(* PLC project steel-plant, Generated TextualNotationConverter 1.0 *)
(* stored: creationDateTime 2025-07-30T12:00:00, modificationDateTime 2025-01-30T12:00:00 *)

FUNCTION_BLOCK ANALOG_IN
  VAR_INPUT
    Name : STRING;
    Description : STRING;
    Raw_Signal : REAL;
    PV_High : REAL;
    PV_Low : REAL;
    Scaling_Slope : REAL;
    Scaling_Offset : REAL;
    Alarm_Enable : BOOL;
  END_VAR
  VAR_OUTPUT
    PV : REAL;
    High_Alarm : BOOL;
    Low_Alarm : BOOL;
    General_Fault : BOOL;
  END_VAR

            
          
END_FUNCTION_BLOCK

FUNCTION_BLOCK PID_BASIC
  VAR_INPUT
    Name : STRING;
    Description : STRING;
    AUTO : BOOL;
    PV : REAL;
    SP : REAL;
    MV_MIN : REAL;
    MV_MAX : REAL;
    X0 : REAL;
    KP : REAL;
    TR : REAL;
    TD : REAL;
    PV_High : REAL;
    PV_Low : REAL;
    Deviation_Limit : REAL;
    Inhibit : BOOL;
  END_VAR
  VAR_OUTPUT
    PV_High_Alarm : BOOL;
    PV_Low_Alarm : BOOL;
    Deviation_Alarm : BOOL;
    XOUT : REAL;
  END_VAR

            
          
END_FUNCTION_BLOCK

FUNCTION_BLOCK RATIO_CONTROL
  VAR_INPUT
    Name : STRING;
    Description : STRING;
    Auto : BOOL;
    PrimaryPV : REAL;
    SecondaryPV : REAL;
    RatioSP : REAL;
    Bias : REAL;
    TrimKp : REAL;
    TrimTi : STRING;
    MV_MIN : REAL;
    MV_MAX : REAL;
    ManOut : REAL;
    Inhibit : BOOL;
  END_VAR
  VAR_OUTPUT
    SlaveSP : REAL;
    ActiveRatio : REAL;
    RatioErr : REAL;
  END_VAR

            
          
END_FUNCTION_BLOCK

FUNCTION_BLOCK VALVE_ELECTRIC
  VAR_INPUT
    Name : STRING;
    Description : STRING;
    Control_Signal : REAL;
    Manual_Mode : BOOL;
    Manual_Position : REAL;
    Open_Limit : REAL;
    Close_Limit : REAL;
    Timeout : STRING;
    Inhibit : BOOL;
  END_VAR
  VAR_OUTPUT
    Valve_Position : REAL;
    Feedback_Pos : REAL;
    Valve_Moving : BOOL;
    Position_Error : BOOL;
    Alarm : BOOL;
  END_VAR

            
          
END_FUNCTION_BLOCK

PROGRAM Section2
  VAR
    FT101_WildFlow_PV : REAL;
    FT102_FluxFlow_PV : REAL;
    TIT101_Temperature_PV : REAL;
    FFIC103_FluxFlowSP : REAL;
    FIC102_ValveCommand : REAL;
  END_VAR
  VAR
    FT-101 : ANALOG_IN;
    FT-102 : ANALOG_IN;
    TIT-101 : ANALOG_IN;
    FV-102 : VALVE_ELECTRIC;
    FIC-102 : PID_BASIC;
    FFIC-103 : RATIO_CONTROL;
  END_VAR
  VAR  (* added by the conversion: wires and edge detectors of the diagram *)
    _OR1_OUT : BOOL;
    _NOT2_OUT : BOOL;
  END_VAR

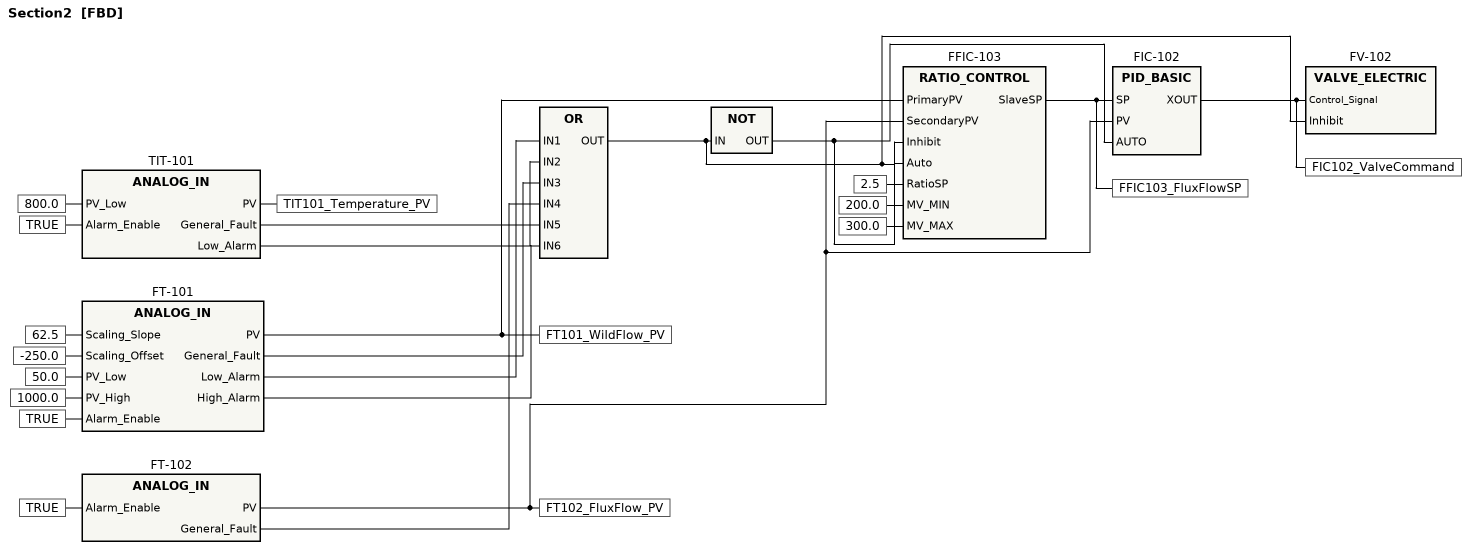
(* FBD diagram, written out as Structured Text *)
FT-101(Scaling_Slope := 62.5, Scaling_Offset := -250.0, PV_Low := 50.0, PV_High := 1000.0, Alarm_Enable := TRUE);
FT-102(Alarm_Enable := TRUE);
TIT-101(PV_Low := 800.0, Alarm_Enable := TRUE);
_OR1_OUT := FT-101.Low_Alarm OR TIT-101.Low_Alarm OR FT-101.General_Fault OR FT-102.General_Fault OR TIT-101.General_Fault OR FT-101.High_Alarm;
_NOT2_OUT := NOT _OR1_OUT;
FFIC-103(PrimaryPV := FT-101.PV, SecondaryPV := FT-102.PV, Inhibit := _OR1_OUT, Auto := _NOT2_OUT, RatioSP := 2.5, MV_MIN := 200.0, MV_MAX := 300.0);
FFIC103_FluxFlowSP := FFIC-103.SlaveSP;
FIC-102(SP := FFIC-103.SlaveSP, PV := FT-102.PV, AUTO := _NOT2_OUT);
FIC102_ValveCommand := FIC-102.XOUT;
FT101_WildFlow_PV := FT-101.PV;
FT102_FluxFlow_PV := FT-102.PV;
TIT101_Temperature_PV := TIT-101.PV;
FV-102(Control_Signal := FIC-102.XOUT, Inhibit := _OR1_OUT);
END_PROGRAM

FUNCTION_BLOCK BOOL_IN
  VAR_INPUT
    Name : STRING;
    Description : STRING;
    Bool_In : BOOL;
    Alarm_OnTrue : BOOL;
    Alarm_OnFalse : BOOL;
    Latch_Enable : BOOL;
    Reset_Latch : BOOL;
  END_VAR
  VAR_OUTPUT
    Bool_Out : BOOL;
    Alarm_Active : BOOL;
    Latched_Status : BOOL;
  END_VAR

            
          
END_FUNCTION_BLOCK

FUNCTION_BLOCK DIGITAL_IN
  VAR_INPUT
    Name : STRING;
    Description : STRING;
    DI_Raw : BOOL;
    DebounceTime : STRING;
    EnableAlarm : BOOL;
  END_VAR
  VAR_OUTPUT
    DI_Out : BOOL;
    Fault_State : BOOL;
  END_VAR

            
          
END_FUNCTION_BLOCK

FUNCTION_BLOCK DUTY_STANDBY
  VAR_INPUT
    Name : STRING;
    Description : STRING;
    Enable : BOOL;
    StartRequest : BOOL;
    AlternateEnable : BOOL;
    ForcePumpA : BOOL;
    ForcePumpB : BOOL;
    DutyElapsed : BOOL;
    MinRunElapsed : BOOL;
    SwitchoverDelayElapsed : BOOL;
    StartTimeoutElapsed : BOOL;
    PumpA_RunFB : BOOL;
    PumpB_RunFB : BOOL;
    PumpA_Fault : BOOL;
    PumpB_Fault : BOOL;
    Reset : BOOL;
    Inhibit : BOOL;
  END_VAR
  VAR_OUTPUT
    CmdPumpA : BOOL;
    CmdPumpB : BOOL;
    ActiveIsA : BOOL;
    SwitchedDueToDuty : BOOL;
    SwitchedDueToFailure : BOOL;
    Alarm_FailedStart_A : BOOL;
    Alarm_FailedStart_B : BOOL;
    Alarm_NoAvailablePump : BOOL;
  END_VAR

            
          
END_FUNCTION_BLOCK

FUNCTION_BLOCK MOTOR_2SPD
  VAR_INPUT
    Name : STRING;
    Description : STRING;
    Start_Cmd : BOOL;
    Stop_Cmd : BOOL;
    Speed_High_Cmd : BOOL;
    Speed_Low_Cmd : BOOL;
    Inhibit : BOOL;
  END_VAR
  VAR_OUTPUT
    Motor_Start_Out : BOOL;
    FB_Running : BOOL;
    FB_Trip : BOOL;
    FB_HighSpeed : BOOL;
    FB_LowSpeed : BOOL;
    Alarm_Speed_Error : BOOL;
  END_VAR

            
          
END_FUNCTION_BLOCK

FUNCTION_BLOCK MOTOR_ON_OFF
  VAR_INPUT
    Name : STRING;
    Description : STRING;
    Start_Cmd : BOOL;
    Stop_Cmd : BOOL;
    Start_Delay : STRING;
    MinRunTime : STRING;
    Inhibit : BOOL;
  END_VAR
  VAR_OUTPUT
    Motor_Start_Out : BOOL;
    FB_Running : BOOL;
    FB_Trip : BOOL;
    Alarm_Start_Fail : BOOL;
    Alarm_Stop_Fail : BOOL;
  END_VAR

            
          
END_FUNCTION_BLOCK

FUNCTION_BLOCK MOTOR_VSD
  VAR_INPUT
    Name : STRING;
    Description : STRING;
    Start_Cmd : BOOL;
    Stop_Cmd : BOOL;
    Speed_SP : REAL;
    Accel_Ramp : STRING;
    Decel_Ramp : STRING;
    Inhibit : BOOL;
  END_VAR
  VAR_OUTPUT
    Speed_Out : REAL;
    FB_Running : BOOL;
    FB_Fault : BOOL;
    FB_Ready : BOOL;
    FB_ActualSpeed : REAL;
    Alarm_Speed_Deviation : BOOL;
    Alarm_Comm_Fail : BOOL;
  END_VAR

            
          
END_FUNCTION_BLOCK

FUNCTION_BLOCK SPLIT_RANGE
  VAR_INPUT
    Name : STRING;
    Description : STRING;
    IN : REAL;
    Split_Point : REAL;
    Output1_Start : REAL;
    Output1_End : REAL;
    Output2_Start : REAL;
    Output2_End : REAL;
  END_VAR
  VAR_OUTPUT
    OUT1 : REAL;
    OUT2 : REAL;
  END_VAR

            
          
END_FUNCTION_BLOCK

FUNCTION_BLOCK VALVE_ON_OFF
  VAR_INPUT
    Name : STRING;
    Description : STRING;
    Open_Cmd : BOOL;
    Close_Cmd : BOOL;
    Timeout : STRING;
    Inhibit : BOOL;
  END_VAR
  VAR_OUTPUT
    FB_Opened : BOOL;
    FB_Closed : BOOL;
    Valve_Open_Out : BOOL;
    Valve_Close_Out : BOOL;
    Alarm_Position_Error : BOOL;
    Alarm_General : BOOL;
  END_VAR

            
          
END_FUNCTION_BLOCK

FUNCTION_BLOCK VOTING_ANALOG
  VAR_INPUT
    Name : STRING;
    Description : STRING;
    Input1 : REAL;
    Input2 : REAL;
    Input3 : REAL;
    Deviation_Limit : REAL;
    Voting_Scheme : STRING;
    EnableAlarm : BOOL;
    Inhibit : BOOL;
  END_VAR
  VAR_OUTPUT
    Voted_Output : REAL;
    Sensor1_Fault : BOOL;
    Sensor2_Fault : BOOL;
    Sensor3_Fault : BOOL;
    Alarm_Voting_Error : BOOL;
    Healthy_Sensors_Count : INT;
  END_VAR

            
          
END_FUNCTION_BLOCK

PROGRAM Section3
  VAR
    PT-201_VOTE : REAL;
    TT-201_VOTE : REAL;
  END_VAR
  VAR
    PT-201A : ANALOG_IN;
    PT-201B : ANALOG_IN;
    PT-201C : ANALOG_IN;
    TT-201A : ANALOG_IN;
    TT-201B : ANALOG_IN;
    TT-201C : ANALOG_IN;
    CO-201 : VOTING_ANALOG;
    CO-202 : VOTING_ANALOG;
    I-201 : BOOL_IN;
    I-202 : BOOL_IN;
    SI-201 : BOOL_IN;
    SI-202 : BOOL_IN;
    MO-201 : DIGITAL_IN;
    MO-202 : DIGITAL_IN;
    P-201 : MOTOR_ON_OFF;
  END_VAR
  VAR  (* added by the conversion: wires and edge detectors of the diagram *)
    _NOT33_OUT : BOOL;
    _NOT34_OUT : BOOL;
    _NOT35_OUT : BOOL;
    _NOT40_OUT : BOOL;
    _NOT41_OUT : BOOL;
    _NOT42_OUT : BOOL;
  END_VAR

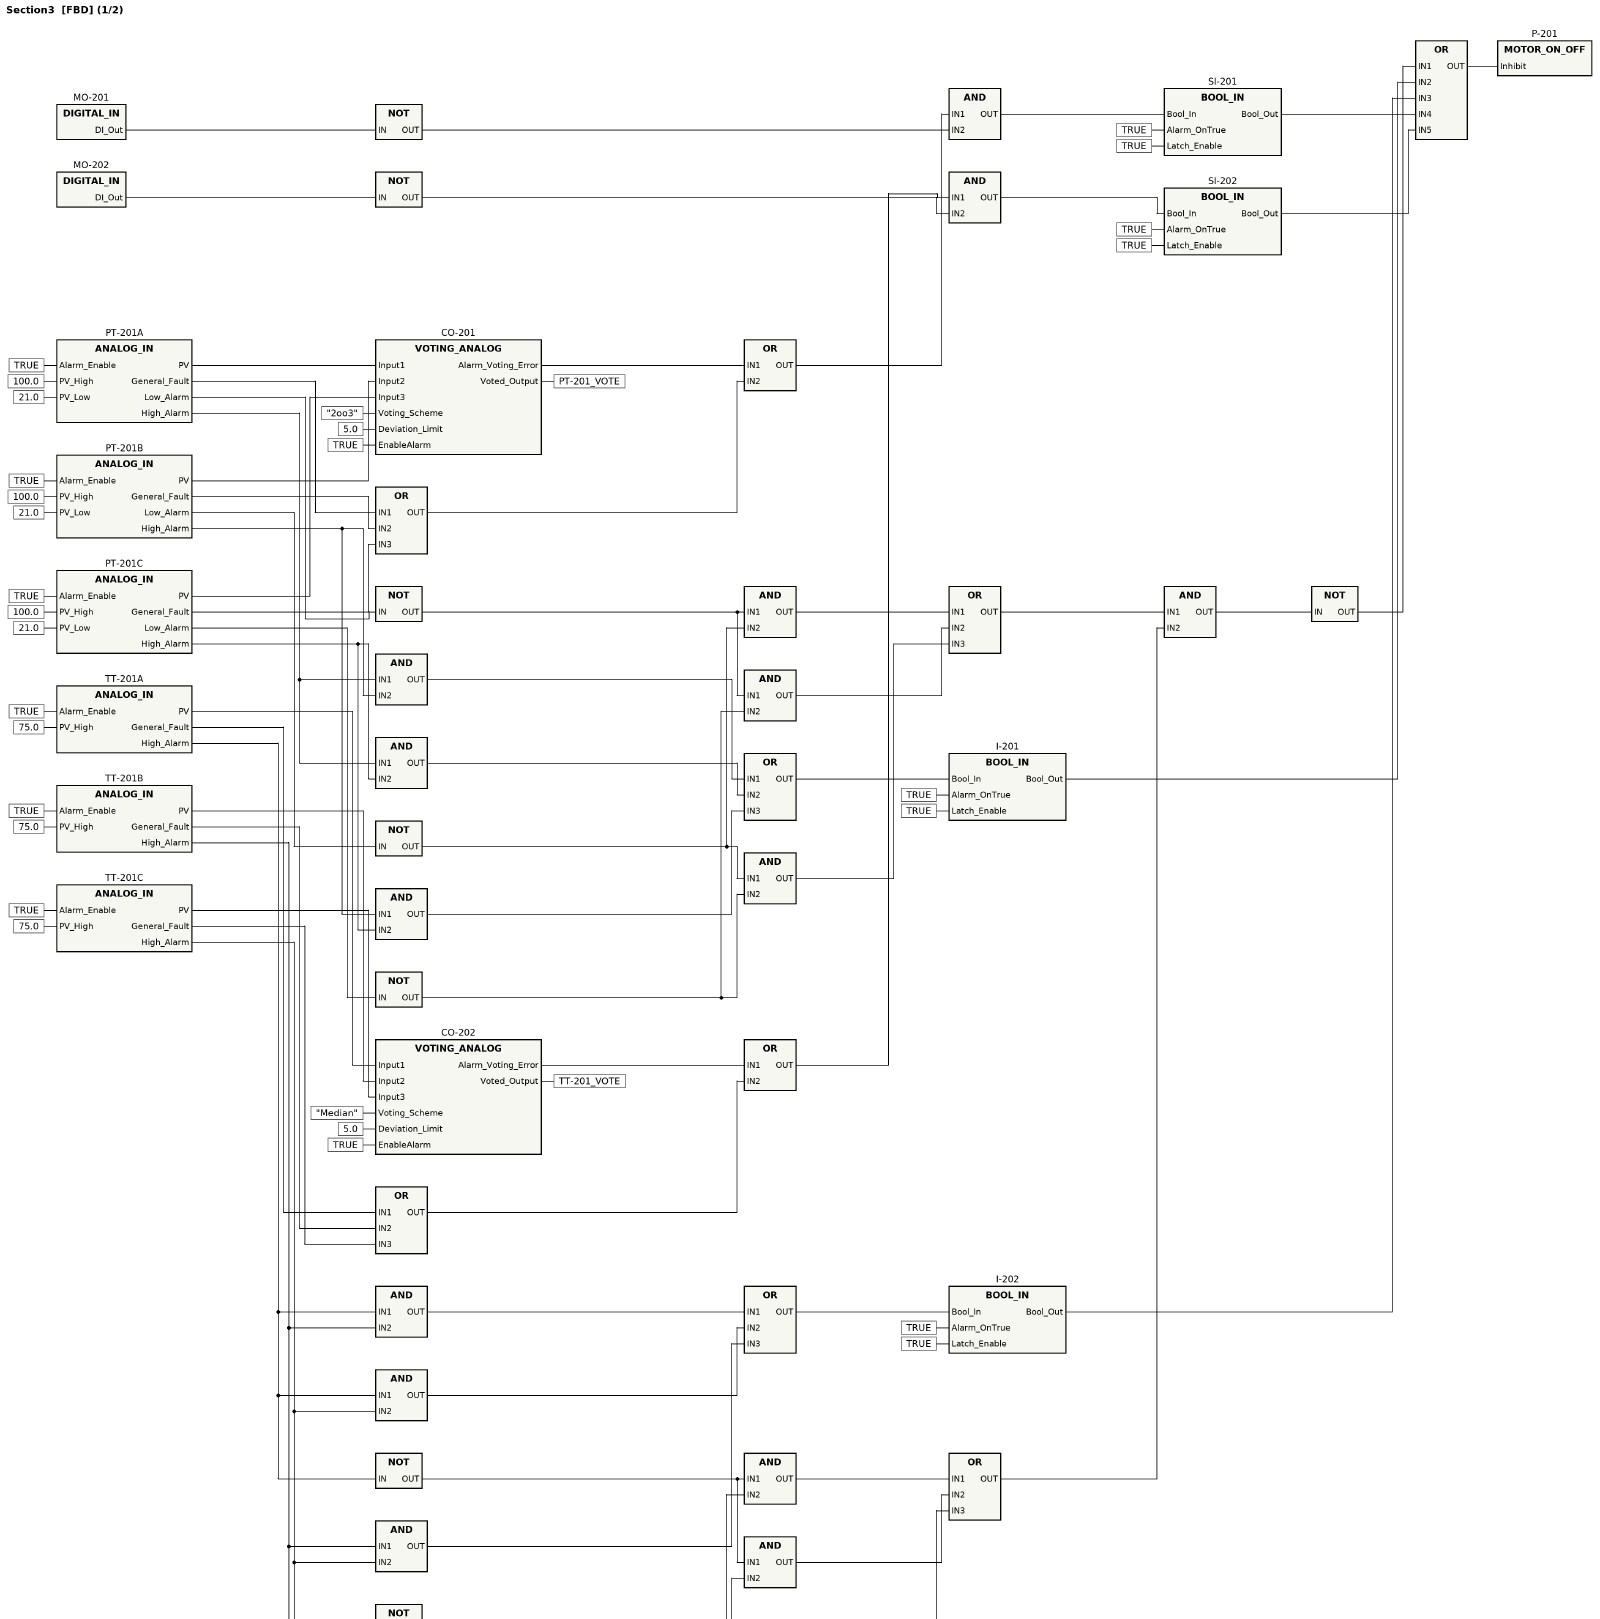
(* FBD diagram, written out as Structured Text *)
PT-201A(Alarm_Enable := TRUE, PV_High := 100.0, PV_Low := 21.0);
PT-201B(Alarm_Enable := TRUE, PV_High := 100.0, PV_Low := 21.0);
PT-201C(Alarm_Enable := TRUE, PV_High := 100.0, PV_Low := 21.0);
CO-201(Input1 := PT-201A.PV, Input2 := PT-201B.PV, Input3 := PT-201C.PV, Voting_Scheme := "2oo3", Deviation_Limit := 5.0, EnableAlarm := TRUE);
PT-201_VOTE := CO-201.Voted_Output;
TT-201A(Alarm_Enable := TRUE, PV_High := 75.0);
TT-201B(Alarm_Enable := TRUE, PV_High := 75.0);
TT-201C(Alarm_Enable := TRUE, PV_High := 75.0);
CO-202(Input1 := TT-201A.PV, Input2 := TT-201B.PV, Input3 := TT-201C.PV, Voting_Scheme := "Median", Deviation_Limit := 5.0, EnableAlarm := TRUE);
TT-201_VOTE := CO-202.Voted_Output;
_NOT33_OUT := NOT PT-201A.Low_Alarm;
_NOT34_OUT := NOT PT-201B.Low_Alarm;
_NOT35_OUT := NOT PT-201C.Low_Alarm;
_NOT40_OUT := NOT TT-201A.High_Alarm;
_NOT41_OUT := NOT TT-201B.High_Alarm;
_NOT42_OUT := NOT TT-201C.High_Alarm;
MO-201();
MO-202();
I-201(Bool_In := PT-201A.High_Alarm AND PT-201B.High_Alarm OR PT-201A.High_Alarm AND PT-201C.High_Alarm OR PT-201B.High_Alarm AND PT-201C.High_Alarm, Alarm_OnTrue := TRUE, Latch_Enable := TRUE);
I-202(Bool_In := TT-201A.High_Alarm AND TT-201B.High_Alarm OR TT-201A.High_Alarm AND TT-201C.High_Alarm OR TT-201B.High_Alarm AND TT-201C.High_Alarm, Alarm_OnTrue := TRUE, Latch_Enable := TRUE);
SI-201(Bool_In := (CO-201.Alarm_Voting_Error OR PT-201A.General_Fault OR PT-201B.General_Fault OR PT-201C.General_Fault) AND NOT MO-201.DI_Out, Alarm_OnTrue := TRUE, Latch_Enable := TRUE);
SI-202(Bool_In := (CO-202.Alarm_Voting_Error OR TT-201A.General_Fault OR TT-201B.General_Fault OR TT-201C.General_Fault) AND NOT MO-202.DI_Out, Alarm_OnTrue := TRUE, Latch_Enable := TRUE);
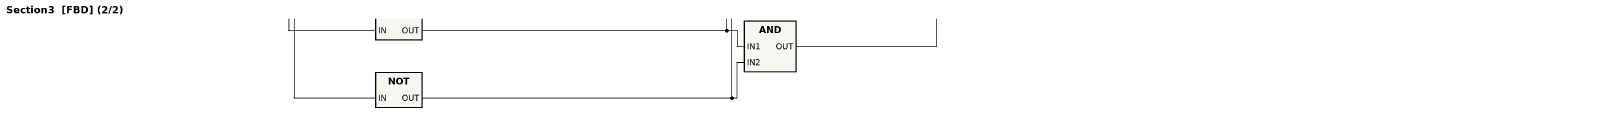
P-201(Inhibit := NOT ((_NOT33_OUT AND _NOT34_OUT OR _NOT33_OUT AND _NOT35_OUT OR _NOT34_OUT AND _NOT35_OUT) AND (_NOT40_OUT AND _NOT41_OUT OR _NOT40_OUT AND _NOT42_OUT OR _NOT41_OUT AND _NOT42_OUT)) OR I-201.Bool_Out OR I-202.Bool_Out OR SI-201.Bool_Out OR SI-202.Bool_Out);
END_PROGRAM

PROGRAM Section4
  VAR
    FFIC303_HotBlastAirFlow_SP : REAL;
    FT301_PulverizedCoalFlow_PV : REAL;
    PT301_FurnacePressure_PV : REAL;
    TT301_HotBlastAirTemperature_PV : REAL;
    HotBlastAirFlow_PV : REAL;
  END_VAR
  VAR
    FT-301 : ANALOG_IN;
    PT-301 : ANALOG_IN;
    TT-301 : ANALOG_IN;
    FFIC-303 : RATIO_CONTROL;
    FIC-302 : PID_BASIC;
    FV-302 : VALVE_ELECTRIC;
  END_VAR
  VAR  (* added by the conversion: wires and edge detectors of the diagram *)
    _OR110_OUT : BOOL;
    _OR115_OUT : BOOL;
  END_VAR

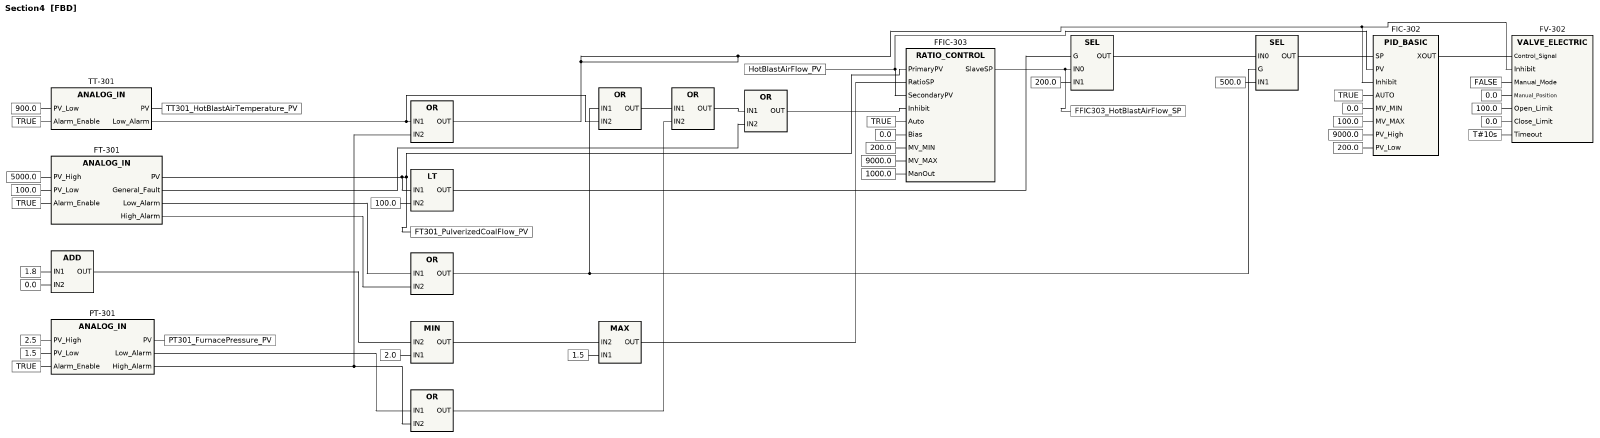
(* FBD diagram, written out as Structured Text *)
FT-301(PV_High := 5000.0, PV_Low := 100.0, Alarm_Enable := TRUE);
_OR110_OUT := FT-301.Low_Alarm OR FT-301.High_Alarm;
TT-301(PV_Low := 900.0, Alarm_Enable := TRUE);
PT-301(PV_High := 2.5, PV_Low := 1.5, Alarm_Enable := TRUE);
FFIC-303(PrimaryPV := FT-301.PV, RatioSP := MAX(MIN(1.8 + 0.0, 2.0), 1.5), SecondaryPV := HotBlastAirFlow_PV, Inhibit := _OR110_OUT OR TT-301.Low_Alarm OR PT-301.Low_Alarm OR PT-301.High_Alarm OR FT-301.General_Fault, Auto := TRUE, Bias := 0.0, MV_MIN := 200.0, MV_MAX := 9000.0, ManOut := 1000.0);
FFIC303_HotBlastAirFlow_SP := FFIC-303.SlaveSP;
FT301_PulverizedCoalFlow_PV := FT-301.PV;
PT301_FurnacePressure_PV := PT-301.PV;
TT301_HotBlastAirTemperature_PV := TT-301.PV;
_OR115_OUT := TT-301.Low_Alarm OR PT-301.High_Alarm;
FIC-302(SP := SEL(SEL(FT-301.PV < 100.0, FFIC-303.SlaveSP, 200.0), _OR110_OUT, 500.0), PV := HotBlastAirFlow_PV, Inhibit := _OR115_OUT, AUTO := TRUE, MV_MIN := 0.0, MV_MAX := 100.0, PV_High := 9000.0, PV_Low := 200.0);
FV-302(Control_Signal := FIC-302.XOUT, Inhibit := _OR115_OUT, Manual_Mode := FALSE, Manual_Position := 0.0, Open_Limit := 100.0, Close_Limit := 0.0, Timeout := T#10s);
END_PROGRAM

PROGRAM Section5
  VAR
    TT_401_V_Voted_Temp : REAL;
  END_VAR
  VAR
    FT-401 : ANALOG_IN;
    PT-401A : ANALOG_IN;
    PT-401B : ANALOG_IN;
    PT-401C : ANALOG_IN;
    TT-401A : ANALOG_IN;
    TT-401B : ANALOG_IN;
    TT-401C : ANALOG_IN;
    TT-401-V : VOTING_ANALOG;
    BOF-402 : VALVE_ELECTRIC;
    I-401 : BOOL_IN;
    DA-401 : BOOL_IN;
    FA-401 : BOOL_IN;
  END_VAR
  VAR  (* added by the conversion: wires and edge detectors of the diagram *)
    _NOT164_OUT : BOOL;
    _NOT166_OUT : BOOL;
    _NOT168_OUT : BOOL;
  END_VAR

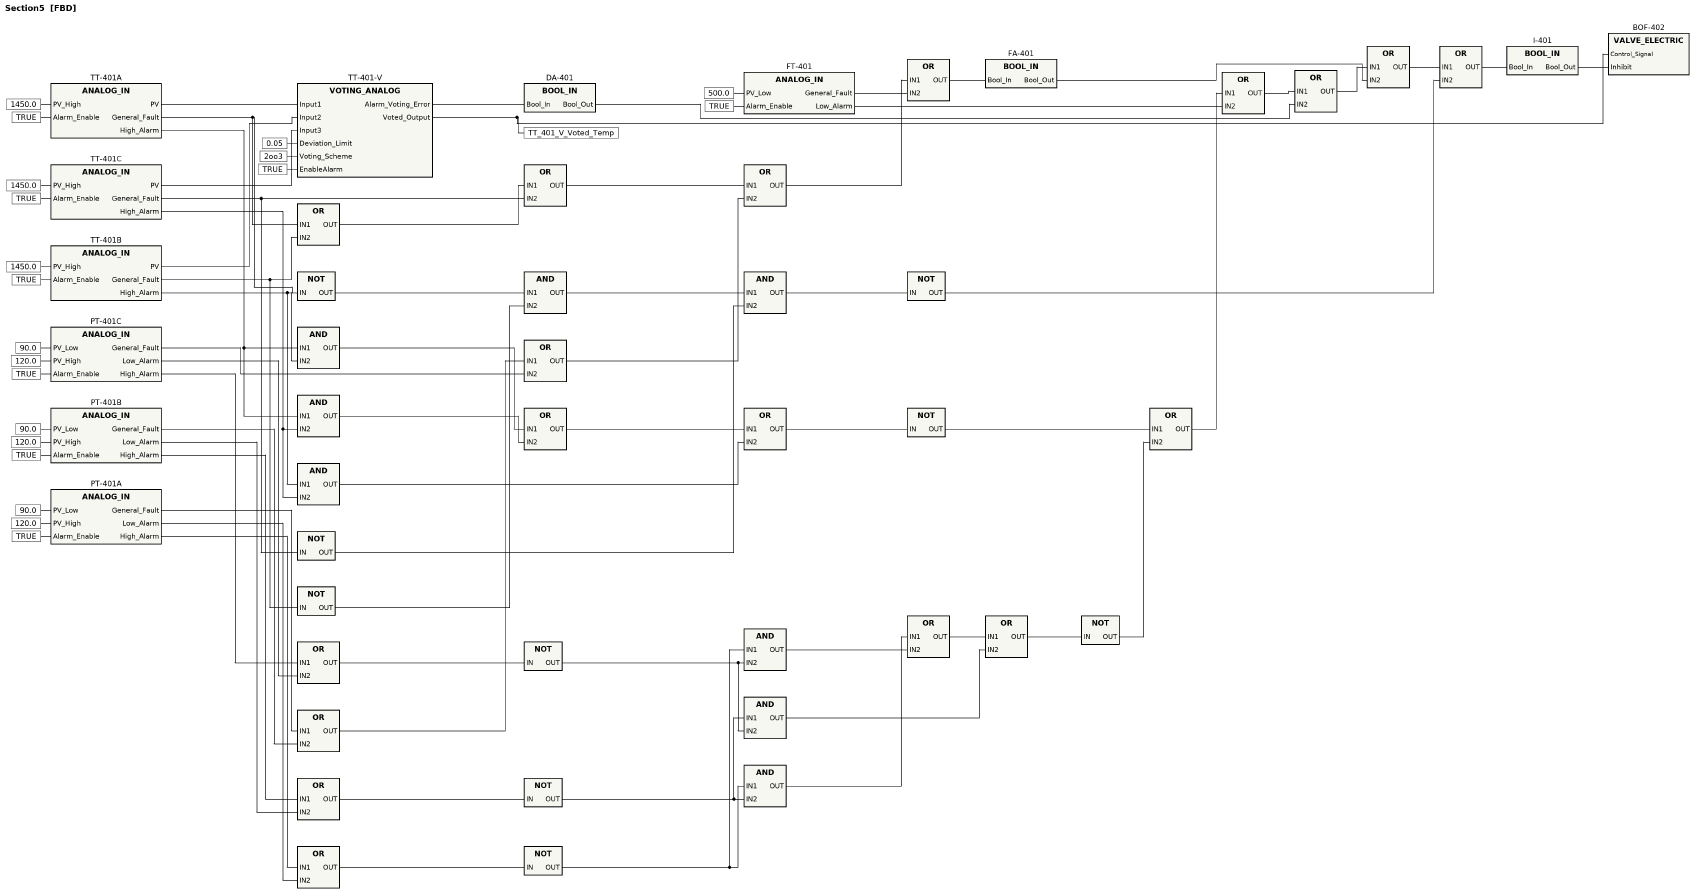
(* FBD diagram, written out as Structured Text *)
TT-401A(PV_High := 1450.0, Alarm_Enable := TRUE);
TT-401B(PV_High := 1450.0, Alarm_Enable := TRUE);
TT-401C(PV_High := 1450.0, Alarm_Enable := TRUE);
TT-401-V(Input1 := TT-401A.PV, Input2 := TT-401B.PV, Input3 := TT-401C.PV, Deviation_Limit := 0.05, Voting_Scheme := 2oo3, EnableAlarm := TRUE);
TT_401_V_Voted_Temp := TT-401-V.Voted_Output;
PT-401A(PV_Low := 90.0, PV_High := 120.0, Alarm_Enable := TRUE);
_NOT164_OUT := NOT (PT-401A.High_Alarm OR PT-401A.Low_Alarm);
PT-401B(PV_Low := 90.0, PV_High := 120.0, Alarm_Enable := TRUE);
_NOT166_OUT := NOT (PT-401B.High_Alarm OR PT-401B.Low_Alarm);
PT-401C(PV_Low := 90.0, PV_High := 120.0, Alarm_Enable := TRUE);
_NOT168_OUT := NOT (PT-401C.High_Alarm OR PT-401C.Low_Alarm);
FT-401(PV_Low := 500.0, Alarm_Enable := TRUE);
DA-401(Bool_In := TT-401-V.Alarm_Voting_Error);
FA-401(Bool_In := TT-401A.General_Fault OR TT-401B.General_Fault OR TT-401C.General_Fault OR PT-401A.General_Fault OR PT-401B.General_Fault OR PT-401C.General_Fault OR FT-401.General_Fault);
I-401(Bool_In := NOT (TT-401A.High_Alarm AND TT-401B.High_Alarm OR TT-401A.High_Alarm AND TT-401C.High_Alarm OR TT-401B.High_Alarm AND TT-401C.High_Alarm) OR NOT (_NOT164_OUT AND _NOT166_OUT OR _NOT164_OUT AND _NOT168_OUT OR _NOT166_OUT AND _NOT168_OUT) OR FT-401.Low_Alarm OR DA-401.Bool_Out OR FA-401.Bool_Out OR NOT (NOT TT-401A.General_Fault AND NOT TT-401B.General_Fault AND NOT TT-401C.General_Fault));
BOF-402(Control_Signal := TT-401-V.Voted_Output, Inhibit := I-401.Bool_Out);
END_PROGRAM

PROGRAM Section6
  VAR
    TT_501_PV : REAL;
    PT_501_PV : REAL;
    SM_501_EA_POS_PV : REAL;
    SM_501_LID_POS : BOOL;
    TT_501_MV : REAL;
    SM_501_EA : REAL;
  END_VAR
  VAR
    TT-501 : ANALOG_IN;
    PT-501 : ANALOG_IN;
    SM-501.EA_POS : ANALOG_IN;
    SM-501.LID_POS : BOOL_IN;
    SM-501 : VALVE_ELECTRIC;
    TT-501_LOOP : PID_BASIC;
  END_VAR
  VAR  (* added by the conversion: wires and edge detectors of the diagram *)
    _OR231_OUT : BOOL;
  END_VAR

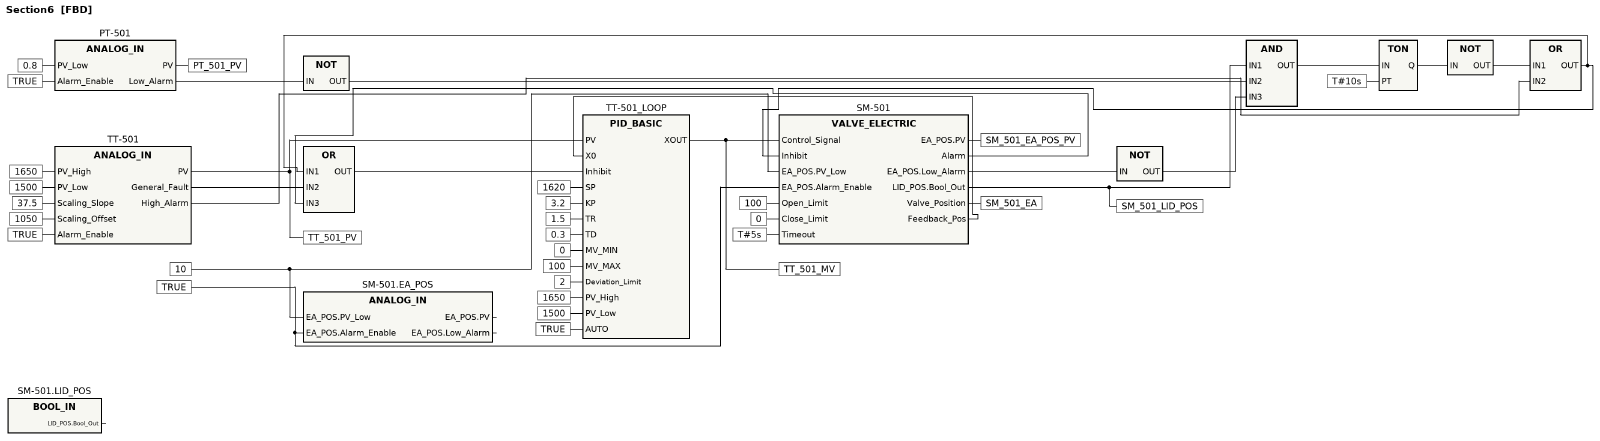
(* FBD diagram, written out as Structured Text *)
PT-501(PV_Low := 0.8, Alarm_Enable := TRUE);
PT_501_PV := PT-501.PV;
TT-501(PV_High := 1650, PV_Low := 1500, Scaling_Slope := 37.5, Scaling_Offset := 1050, Alarm_Enable := TRUE);
_OR231_OUT := NOT TON(SM-501.LID_POS.Bool_Out AND NOT PT-501.Low_Alarm AND NOT SM-501.EA_POS.Low_Alarm, T#10s) OR TT-501.High_Alarm;
TT-501_LOOP(PV := TT-501.PV, X0 := SM-501.Feedback_Pos, Inhibit := _OR231_OUT OR TT-501.General_Fault OR SM-501.Alarm, SP := 1620, KP := 3.2, TR := 1.5, TD := 0.3, MV_MIN := 0, MV_MAX := 100, Deviation_Limit := 2, PV_High := 1650, PV_Low := 1500, AUTO := TRUE);
SM-501(Control_Signal := TT-501_LOOP.XOUT, Inhibit := _OR231_OUT, EA_POS.PV_Low := 10, EA_POS.Alarm_Enable := TRUE, Open_Limit := 100, Close_Limit := 0, Timeout := T#5s);
SM_501_EA := SM-501.Valve_Position;
SM_501_EA_POS_PV := SM-501.EA_POS.PV;
SM_501_LID_POS := SM-501.LID_POS.Bool_Out;
TT_501_MV := TT-501_LOOP.XOUT;
TT_501_PV := TT-501.PV;
SM-501.EA_POS(EA_POS.PV_Low := 10, EA_POS.Alarm_Enable := TRUE);
SM-501.LID_POS();
END_PROGRAM

PROGRAM Section7
  VAR
    LIT101_MoldLevel_PV_mm : REAL;
    FT601_CoolingWaterFlow_PV_m3ph : REAL;
    TT601_MoldTemp_PV_degC : REAL;
    LIC101_ValveCommand_Percent : REAL;
    MV101_ValvePosition_Percent : REAL;
  END_VAR
  VAR
    LIT-101 : ANALOG_IN;
    FT-601 : ANALOG_IN;
    TT-601 : ANALOG_IN;
    LIC-101 : PID_BASIC;
    MV-101 : VALVE_ELECTRIC;
  END_VAR
  VAR  (* added by the conversion: wires and edge detectors of the diagram *)
    _OR267_OUT : BOOL;
  END_VAR

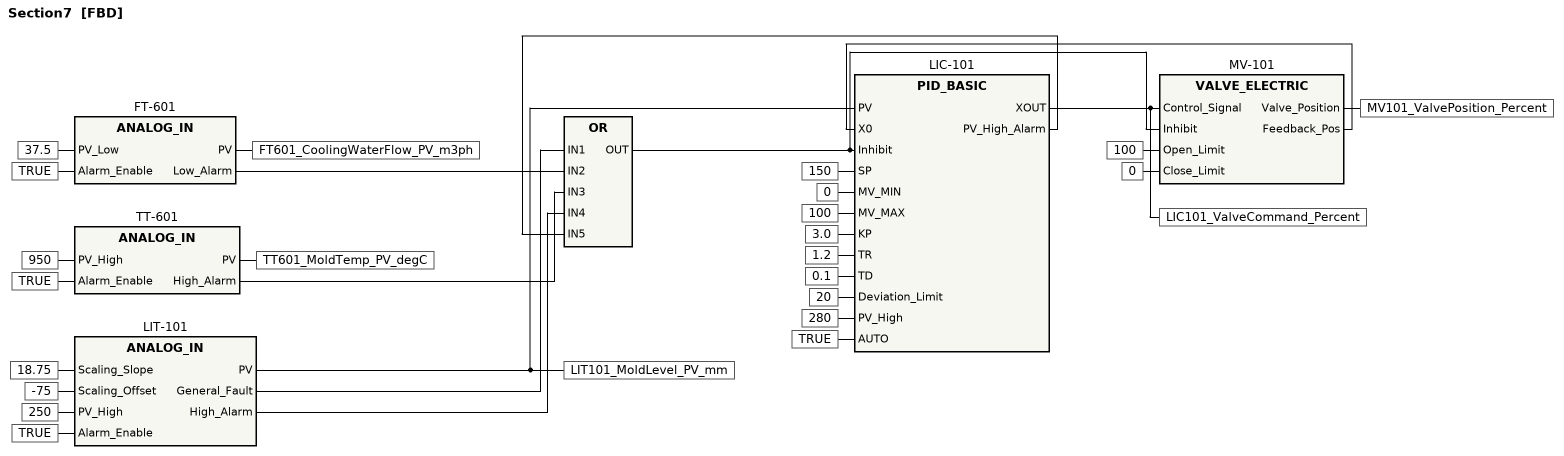
(* FBD diagram, written out as Structured Text *)
FT-601(PV_Low := 37.5, Alarm_Enable := TRUE);
FT601_CoolingWaterFlow_PV_m3ph := FT-601.PV;
LIT-101(Scaling_Slope := 18.75, Scaling_Offset := -75, PV_High := 250, Alarm_Enable := TRUE);
TT-601(PV_High := 950, Alarm_Enable := TRUE);
_OR267_OUT := LIT-101.General_Fault OR FT-601.Low_Alarm OR TT-601.High_Alarm OR LIT-101.High_Alarm OR LIC-101.PV_High_Alarm;
MV-101(Control_Signal := LIC-101.XOUT, Inhibit := _OR267_OUT, Open_Limit := 100, Close_Limit := 0);
LIC-101(PV := LIT-101.PV, X0 := MV-101.Feedback_Pos, Inhibit := _OR267_OUT, SP := 150, MV_MIN := 0, MV_MAX := 100, KP := 3.0, TR := 1.2, TD := 0.1, Deviation_Limit := 20, PV_High := 280, AUTO := TRUE);
LIC101_ValveCommand_Percent := LIC-101.XOUT;
LIT101_MoldLevel_PV_mm := LIT-101.PV;
MV101_ValvePosition_Percent := MV-101.Valve_Position;
TT601_MoldTemp_PV_degC := TT-601.PV;
END_PROGRAM

PROGRAM Section8
  VAR
    FT701_FuelFlow_PV : REAL;
    FT702_AirFlow_SP : REAL;
    FT702_AirFlow_PV : REAL;
    TT701_FurnaceTemp_PV : REAL;
    FFIC701_Bias : REAL;
    BURNER_STATUS : BOOL;
  END_VAR
  VAR
    FT-701 : ANALOG_IN;
    FT-702 : ANALOG_IN;
    TT-701 : ANALOG_IN;
    FIC-702 : PID_BASIC;
    FV-702 : VALVE_ELECTRIC;
    FFIC-701 : RATIO_CONTROL;
    BLS-701 : BOOL_IN;
    ALM-701 : DIGITAL_IN;
    ALM-702 : DIGITAL_IN;
    ALM-703 : DIGITAL_IN;
    ALM-704 : DIGITAL_IN;
  END_VAR
  VAR  (* added by the conversion: wires and edge detectors of the diagram *)
    _OR298_OUT : BOOL;
  END_VAR

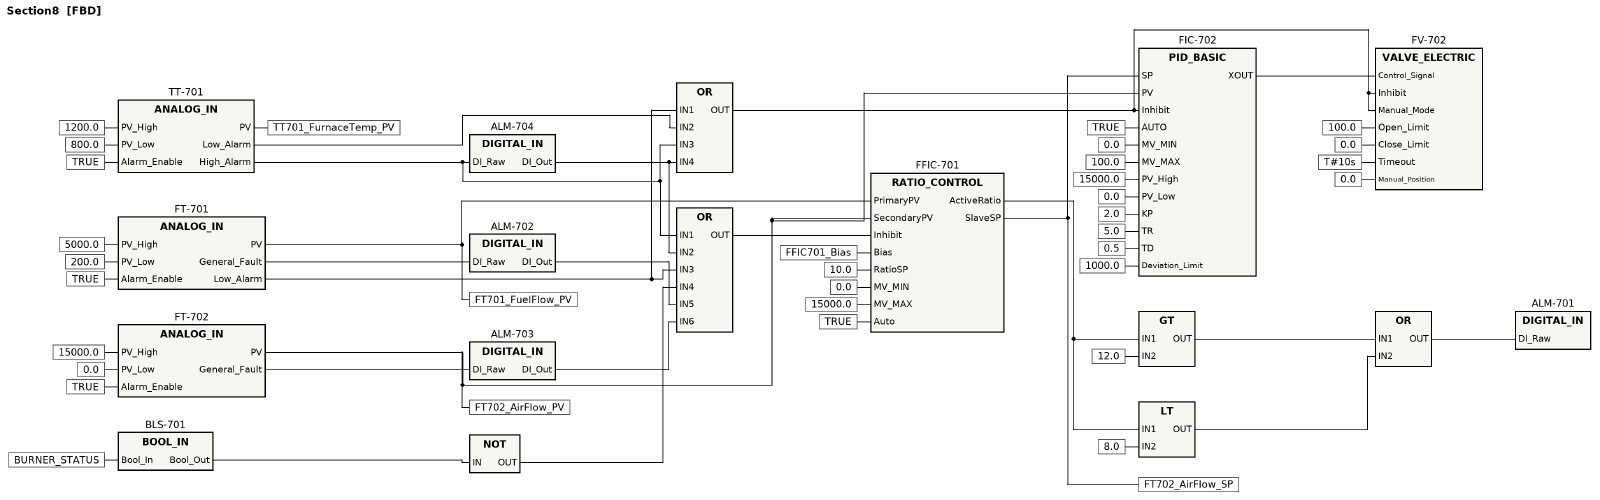
(* FBD diagram, written out as Structured Text *)
FT-701(PV_High := 5000.0, PV_Low := 200.0, Alarm_Enable := TRUE);
FT701_FuelFlow_PV := FT-701.PV;
FT-702(PV_High := 15000.0, PV_Low := 0.0, Alarm_Enable := TRUE);
FT702_AirFlow_PV := FT-702.PV;
TT-701(PV_High := 1200.0, PV_Low := 800.0, Alarm_Enable := TRUE);
ALM-704(DI_Raw := TT-701.High_Alarm);
BLS-701(Bool_In := BURNER_STATUS);
ALM-702(DI_Raw := FT-701.General_Fault);
ALM-703(DI_Raw := FT-702.General_Fault);
FFIC-701(PrimaryPV := FT-701.PV, SecondaryPV := FT-702.PV, Inhibit := TT-701.High_Alarm OR ALM-704.DI_Out OR FT-701.Low_Alarm OR NOT BLS-701.Bool_Out OR ALM-702.DI_Out OR ALM-703.DI_Out, Bias := FFIC701_Bias, RatioSP := 10.0, MV_MIN := 0.0, MV_MAX := 15000.0, Auto := TRUE);
FT702_AirFlow_SP := FFIC-701.SlaveSP;
TT701_FurnaceTemp_PV := TT-701.PV;
_OR298_OUT := FT-701.Low_Alarm OR TT-701.Low_Alarm OR TT-701.High_Alarm OR ALM-704.DI_Out;
FIC-702(SP := FFIC-701.SlaveSP, PV := FT-702.PV, Inhibit := _OR298_OUT, AUTO := TRUE, MV_MIN := 0.0, MV_MAX := 100.0, PV_High := 15000.0, PV_Low := 0.0, KP := 2.0, TR := 5.0, TD := 0.5, Deviation_Limit := 1000.0);
FV-702(Control_Signal := FIC-702.XOUT, Inhibit := _OR298_OUT, Manual_Mode := _OR298_OUT, Open_Limit := 100.0, Close_Limit := 0.0, Timeout := T#10s, Manual_Position := 0.0);
ALM-701(DI_Raw := FFIC-701.ActiveRatio > 12.0 OR FFIC-701.ActiveRatio < 8.0);
END_PROGRAM

PROGRAM Section9
  VAR
    FIC802_AirFlow_SP_FromRatio : REAL;
    FFIC801_ActiveAirToGasRatio : REAL;
    FT801_BFG_Flow_PV : REAL;
    FT802_Air_Flow_PV : REAL;
    PT801_BFG_Pressure_PV : REAL;
    AL801_HighRatio_SP : REAL;
    AL802_LowRatio_SP : REAL;
    AL801_HighRatio_Alarm : BOOL;
    AL802_LowRatio_Alarm : BOOL;
    AL803_FT801_Fault_Alarm : BOOL;
    AL804_PT801_Fault_Alarm : BOOL;
  END_VAR
  VAR
    AL-801 : ANALOG_IN;
    AL-802 : ANALOG_IN;
    AL-803 : ANALOG_IN;
    AL-804 : ANALOG_IN;
    FT-801 : ANALOG_IN;
    FT-802 : ANALOG_IN;
    PT-801 : ANALOG_IN;
    FFIC-801 : RATIO_CONTROL;
    FIC-802 : PID_BASIC;
    FV-802 : VALVE_ELECTRIC;
    HighRatio_TON : TON;
  END_VAR
  VAR  (* added by the conversion: wires and edge detectors of the diagram *)
    _OR352_OUT : BOOL;
    _OR348_OUT : BOOL;
  END_VAR

(* FBD diagram, written out as Structured Text *)
FT-801(Scaling_Slope := 6.25, Scaling_Offset := -25.0, PV_Low := 100.0, PV_High := 5000.0, Alarm_Enable := TRUE);
FT-802(Scaling_Slope := 6.25, Scaling_Offset := -25.0, PV_Low := 0.0, PV_High := 6000.0, Alarm_Enable := TRUE);
PT-801(Scaling_Slope := 6.25, Scaling_Offset := -25.0, PV_Low := 0.5, PV_High := 2.0, Alarm_Enable := TRUE);
_OR352_OUT := FT-801.Low_Alarm OR FT-801.General_Fault OR PT-801.General_Fault;
_OR348_OUT := PT-801.High_Alarm OR PT-801.Low_Alarm;
FFIC-801(PrimaryPV := FT-801.PV, SecondaryPV := FT-802.PV, Inhibit := _OR352_OUT OR FT-802.High_Alarm OR _OR348_OUT, RatioSP := 2.5, MV_MIN := 0.0, MV_MAX := 6000.0, Bias := 0.0, TrimKp := 0.0, TrimTi := T#0s, Auto := TRUE);
HighRatio_TON(IN := FFIC-801.ActiveRatio > AL801_HighRatio_SP, PT := T#5s);
AL801_HighRatio_Alarm := HighRatio_TON.Q;
AL802_LowRatio_Alarm := FFIC-801.ActiveRatio < AL802_LowRatio_SP;
AL803_FT801_Fault_Alarm := FT-801.General_Fault;
AL804_PT801_Fault_Alarm := PT-801.General_Fault;
FFIC801_ActiveAirToGasRatio := FFIC-801.ActiveRatio;
FIC802_AirFlow_SP_FromRatio := FFIC-801.SlaveSP;
FT801_BFG_Flow_PV := FT-801.PV;
FT802_Air_Flow_PV := FT-802.PV;
PT801_BFG_Pressure_PV := PT-801.PV;
AL-801(Alarm_Enable := TRUE);
AL-802(Alarm_Enable := TRUE);
AL-803();
AL-804();
FIC-802(SP := FFIC-801.SlaveSP, PV := FT-802.PV, Inhibit := _OR352_OUT, AUTO := TRUE, MV_MIN := 0.0, MV_MAX := 100.0, PV_Low := 0.0, PV_High := 6000.0, X0 := 50.0);
FV-802(Control_Signal := FIC-802.XOUT, Inhibit := _OR348_OUT, Manual_Position := 50.0);
(* drawn but not wired to any output: 3.0, 2.0 *)
END_PROGRAM

CONFIGURATION Config0
  RESOURCE Res0 ON PLC
    TASK task0(INTERVAL := T#20ms, PRIORITY := 0);
    PROGRAM instance0 WITH task0 : Section2;
    PROGRAM instance_1 WITH task0 : Section3;
    PROGRAM instance_2 WITH task0 : Section4;
    PROGRAM instance_3 WITH task0 : Section5;
    PROGRAM instance_4 WITH task0 : Section6;
    PROGRAM instance_5 WITH task0 : Section7;
    PROGRAM instance_6 WITH task0 : Section8;
    PROGRAM instance_7 WITH task0 : Section9;
  END_RESOURCE
END_CONFIGURATION
